// TwinCAT 3 PLC project HomePLC_AlarmManager
// Title: HomePLC Alarm Manager
// Company: Tom Oyen
// Author: Tom Oyen
// ProjectVersion: 1.0.5
// Description: Alarm manager
// ProgramVersion: 3.1.4024.0
// libraries:
//   HomePLC DIO, * (Tom Oyen)
//   HomePLC Logging, * (Tom Oyen)
//   Tc2_Standard, * (Beckhoff Automation GmbH)
//   Tc2_System, * (Beckhoff Automation GmbH)
//   Tc2_Utilities, * (Beckhoff Automation GmbH)
//   Tc3_Module, * (Beckhoff Automation GmbH)
// project tree:
//   DUTs/ E_AlarmManagerStep.TcDUT, E_AlarmState.TcDUT, ST_AlarmManagerHMI.TcDUT
//   / GlobalTextList.TcGTLO, Visualization Manager.TcVMO (not stored)
//   GVLs/ GVL_AlarmManager.TcGVL
//   POUs/ FB_AlarmManager.TcPOU, I_AlarmManager.TcIO
//   POUs/Keypad/DUTs/ E_KeypadState.TcDUT, ST_AlarmKeypadHMI.TcDUT, ST_AlarmKeypadVirtual.TcDUT, ST_LedState.TcDUT
//   POUs/Keypad/ FB_AlarmKeypad.TcPOU, I_AlarmKeypad.TcIO
//   POUs/Sensor/DUTs/ ST_AlarmSensorHMI.TcDUT
//   POUs/Sensor/ FB_AlarmSensor.TcPOU, I_AlarmSensor.TcIO
//   POUs/Siren/DUTs/ ST_AlarmSirenHMI.TcDUT
//   POUs/Siren/ FB_AlarmSiren.TcPOU, I_AlarmSiren.TcIO
//   Project Information/ F_GetCompany.TcPOU, F_GetTitle.TcPOU, F_GetVersion.TcPOU
//   UTIL/ GetDateTime.TcPOU
//   Version/ Global_Version.TcGVL
//   VISUs/ Alarm.TcVIS, Keypad.TcVIS, Siren.TcVIS, Sensor.TcVIS

// ---- DUTs/E_AlarmManagerStep.TcDUT
{attribute 'qualified_only'}
{attribute 'strict'}
TYPE E_AlarmManagerStep :
(
	Init 					:= 0,
	CheckEnable				:= 1,
	
	HardwareCheck			:= 10,
	Enabling				:= 11,
	Enable					:= 12,
	
	CheckSensors			:= 20,
	
	Warn					:= 30,
	WaitForDisableWarn		:= 31,
	SoundAlarm				:= 32,
	WaitForDisableAlarm		:= 33,
	
	Disabling				:= 40,
	Disable					:= 41,
	
	Reset					:= 50
);
END_TYPE

// ---- DUTs/E_AlarmState.TcDUT
{attribute 'qualified_only'}
{attribute 'strict'}
{attribute 'to_string'}
TYPE E_AlarmState :
(
	Off 			:= 0,
	Enabling		:= 1,
	Enabled			:= 2,
	Warning			:= 3,
	Tripped			:= 4,
	Disabling		:= 5
);
END_TYPE

// ---- DUTs/ST_AlarmManagerHMI.TcDUT
TYPE ST_AlarmManagerHMI :
STRUCT
	// General
	nKeypads		: INT;				// Number of keypads
	nSensors		: INT;				// Number of sensors
	nSirens			: INT;				// Number of sirens
	eState			: E_AlarmState;		// Alarm enabled state
	nActiveID		: INT;				// ID of alarm component which was last active
	nActiveReason	: INT;				// Reason why alarm component was active
	
	// Overview
	aSensors		: ARRAY [0..GVL_AlarmManager.nMaxSensors - 1] OF ST_AlarmSensorHMI;
	aSirens			: ARRAY [0..GVL_AlarmManager.nMaxSirens - 1] OF ST_AlarmSirenHMI;
END_STRUCT
END_TYPE

// ---- POUs/Keypad/DUTs/E_KeypadState.TcDUT
{attribute 'qualified_only'}
{attribute 'strict'}
TYPE E_KeypadState :
(
	Init 				:= 0,
	Idle				:= 1,
	InputDetected		:= 2,
	CheckInput			:= 3,
	Reset				:= 4	
);
END_TYPE

// ---- POUs/Keypad/DUTs/ST_AlarmKeypadHMI.TcDUT
TYPE ST_AlarmKeypadHMI :
STRUCT
	sName			: STRING;
	
	bLed1			: BOOL;
	bLed2			: BOOL;
	bLed3			: BOOL;
	bLed4			: BOOL;
	bLed5			: BOOL;
	bLed6			: BOOL;
	
	bBuzzer			: BOOL;
	
	sCode			: STRING;
END_STRUCT
END_TYPE

// ---- POUs/Keypad/DUTs/ST_AlarmKeypadVirtual.TcDUT
TYPE ST_AlarmKeypadVirtual :
STRUCT
	bButton1			: BOOL;
	bButton2			: BOOL;
	bButton3			: BOOL;
	bButton4			: BOOL;
	bButton5			: BOOL;
	bButton6			: BOOL;
END_STRUCT
END_TYPE

// ---- POUs/Keypad/DUTs/ST_LedState.TcDUT
TYPE ST_LedState :
STRUCT
	eLed1	: E_DOCommand;
	eLed2	: E_DOCommand;
	eLed3	: E_DOCommand;
	eLed4	: E_DOCommand;
	eLed5	: E_DOCommand;
	eLed6	: E_DOCommand;
END_STRUCT
END_TYPE

// ---- POUs/Sensor/DUTs/ST_AlarmSensorHMI.TcDUT
TYPE ST_AlarmSensorHMI :
STRUCT
	sName		: STRING;	// Sensor name
	nID			: INT;		// Alarm component ID
	bAlarm		: BOOL;		// True if the sensor detects something
	bTamper		: BOOL;		// True if the sensor is tampered with
	bDisabled	: BOOL;		// True if the sensor is disabled
END_STRUCT
END_TYPE

// ---- POUs/Siren/DUTs/ST_AlarmSirenHMI.TcDUT
TYPE ST_AlarmSirenHMI :
STRUCT
	sName		: STRING;	// Siren name
	nID			: INT;		// Alarm component ID
	bSiren		: BOOL;		// True if the siren is on
	bLight		: BOOL;		// True if the light is on
	bTamper		: BOOL;		// True if the siren is tampered with
END_STRUCT
END_TYPE

// ---- GVLs/GVL_AlarmManager.TcGVL
{attribute 'qualified_only'}
VAR_GLOBAL CONSTANT
	nMaxKeypads		: INT := 5;										// Maximum number of keypads
	nMaxSirens		: INT := 5;										// Maximum number of sirens
	nMaxSensors		: INT := 10;									// Maximum number of sensors
	sCode			: STRING := '1234';								// Configured alarm code
END_VAR

// ---- Version/Global_Version.TcGVL
{attribute 'TcGenerated'}
{attribute 'no-analysis'}
{attribute 'linkalways'}
// This function has been automatically generated from the project information.
VAR_GLOBAL CONSTANT
	{attribute 'const_non_replaced'}
	stLibVersion_HomePLC_Alarm_Manager : ST_LibVersion := (iMajor := 1, iMinor := 0, iBuild := 5, iRevision := 0, nFlags := 0, sVersion := '1.0.5');
END_VAR

// ---- POUs/I_AlarmManager.TcIO
// Alarm manager interface
INTERFACE I_AlarmManager

// Add a keypad to the alarm manager
METHOD AddKeypad
VAR_INPUT
	IKeypad		: I_AlarmKeypad;		// Keypad interface
END_VAR
END_METHOD

// Add an alarm sensor to the alarm manager
METHOD AddSensor
VAR_INPUT
	ISensor		: I_AlarmSensor;		// Alarm sensor interface
END_VAR
END_METHOD

// Add a siren to the alarm manager
METHOD AddSiren
VAR_INPUT
	ISiren		: I_AlarmSiren;		// Siren interface
END_VAR
END_METHOD

END_INTERFACE

// ---- POUs/Keypad/I_AlarmKeypad.TcIO
// Alarm keypad interface
INTERFACE I_AlarmKeypad

// Returns true if the user input code equals the configured code
METHOD CheckCode : BOOL
END_METHOD

// Run this method every cycle
METHOD Execute
END_METHOD

// Returns the HMI data
PROPERTY HmiData : ST_AlarmKeypadHMI
GET
END_GET
END_PROPERTY

// Returns the keypad name
PROPERTY Name : STRING
GET
END_GET
END_PROPERTY

// Call this method once when the alarm state is changed
METHOD SetAlarmState
VAR_INPUT
	eAlarmState			: E_AlarmState;		// Alarm state
END_VAR
END_METHOD

// Set the buzzer command
METHOD SetBuzzer
VAR_INPUT
	eCommand	: E_DOCommand;
END_VAR
END_METHOD

// Set the keypad configured code
METHOD SetConfiguredCode
VAR_INPUT
	sCode	:	STRING;		// Configured code
END_VAR
END_METHOD

// Returns true if the buzzer needs to sound to indicate the alarm status
PROPERTY SoundBuzzer : BOOL
GET
END_GET
END_PROPERTY

END_INTERFACE

// ---- POUs/Sensor/I_AlarmSensor.TcIO
// Alarm sensor interface
INTERFACE I_AlarmSensor

// Returns true if the sensor detects something (as long as something is detected)
PROPERTY Alarm : BOOL
GET
END_GET
END_PROPERTY

// Returns true when the sensor is triggered (one cycle)
PROPERTY AlarmTrigger : BOOL
GET
END_GET
END_PROPERTY

// Run this method every cycle
METHOD Execute
END_METHOD

// Returns the HMI data
PROPERTY HmiData : ST_AlarmSensorHMI
GET
END_GET
END_PROPERTY

// Get the alarm component ID of the sensor
PROPERTY ID : INT
GET
END_GET
END_PROPERTY

// Gets the outputs to turn on when the sensor is triggered
PROPERTY OutputsOnDetect : ARRAY [0..9] OF I_DigitalOut
GET
END_GET
END_PROPERTY

// Number of outputs to enable when the sensor is triggered
PROPERTY OutputsOnDetectSize : INT
GET
END_GET
END_PROPERTY

// Set the sensor disable state
METHOD SetDisableState
VAR_INPUT
	bDisable	: BOOL;		// Set to true to disable the sensor
END_VAR
END_METHOD

// Returns true when the sensor is tampered with (as long as the sensor is tampered with)
PROPERTY Tamper : BOOL
GET
END_GET
END_PROPERTY

// Returns true when the tamper sensor is triggered (one cycle)
PROPERTY TamperTrigger : BOOL
GET
END_GET
END_PROPERTY

// Returs true if the user is warned before the alarm is set off
PROPERTY WarnFirst : BOOL
GET
END_GET
END_PROPERTY

END_INTERFACE

// ---- POUs/Siren/I_AlarmSiren.TcIO
INTERFACE I_AlarmSiren

// Run this method every cycle
METHOD Execute
END_METHOD

// Returns the HMI data
PROPERTY HmiData : ST_AlarmSirenHMI
GET
END_GET
END_PROPERTY

// Get the alarm component ID of the siren
PROPERTY ID : INT
GET
END_GET
END_PROPERTY

// Set siren light
METHOD SetLight
VAR_INPUT
	eCommand	: E_DOCommand;		// Siren digital output command
END_VAR
END_METHOD

// Set siren sound
METHOD SetSound
VAR_INPUT
	eCommand	: E_DOCommand;		// Siren sound digital output command
END_VAR
END_METHOD

// Returns true when the siren is tampered with (as long as the siren is tampered with)
PROPERTY Tamper : BOOL
GET
END_GET
END_PROPERTY

// Returns true when the tamper sensor is triggered (one cycle)
PROPERTY TamperTrigger : BOOL
GET
END_GET
END_PROPERTY

END_INTERFACE

// ---- POUs/FB_AlarmManager.TcPOU
// Alarm manager
{attribute 'reflection'} 
FUNCTION_BLOCK FB_AlarmManager IMPLEMENTS I_AlarmManager
VAR
	aKeypads				: ARRAY [0..GVL_AlarmManager.nMaxKeypads - 1] OF I_AlarmKeypad;		// Keypads
	nKeypads				: INT;																// Number of keypads
	
	aSensors				: ARRAY [0..GVL_AlarmManager.nMaxSensors - 1] OF I_AlarmSensor;		// Alarm sensors
	nSensors				: INT;																// Number of alarm sensors
	
	aSirens					: ARRAY [0..GVL_AlarmManager.nMaxSirens - 1] OF I_AlarmSiren;		// Alarm sirens
	nSirens					: INT;																// Number of alarm sirens
	
	eState					: E_AlarmState;														// Alarm state
	
	bEnabling		AT %Q*	: BOOL;																// Alarm enabling (can be read externally)
	bEnabled		AT %Q*	: BOOL;																// Alarm enabled (can be read externally)
	nState			AT %Q*	: INT;																// Alarm state number (can be read externally)
	nActiveID		AT %Q*	: INT;																// Alarm component ID that tripped alarm (can be read externally)
	nActiveReason	AT %Q*	: INT;																// ID reason alarm was tripped (can be read externally)
	
	fbLogger				: class_Tc3EventLogger;												// Logging FB

	// Use attributes to copy instance name to sName
	{attribute 'instance-path'} 
    {attribute 'noinit'} 
    sName					: STRING; 															// Instance name
	
	stHMI					: ST_AlarmManagerHMI;												// HMI data
END_VAR

// Add a keypad to the alarm manager
METHOD AddKeypad
VAR_INPUT
	IKeypad		: I_AlarmKeypad;		// Keypad interface
END_VAR
// Add keypad
aKeypads[nKeypads] := IKeypad;
nKeypads := nKeypads + 1;
END_METHOD

// Add an alarm sensor to the alarm manager
METHOD AddSensor
VAR_INPUT
	ISensor		: I_AlarmSensor;		// Alarm sensor interface
END_VAR
// Add alarm sensor
aSensors[nSensors] := ISensor;
nSensors := nSensors + 1;
END_METHOD

// Add a siren to the alarm manager
METHOD AddSiren
VAR_INPUT
	ISiren		: I_AlarmSiren;		// Siren interface
END_VAR
// Add siren
aSirens[nSirens] := ISiren;
nSirens := nSirens + 1;
END_METHOD

// Run this method every cycle
METHOD Execute
VAR_INST
	eStep						: E_AlarmManagerStep;	// Alarm manager state machine step
	eStepPrev					: E_AlarmManagerStep;	// Alarm manager state machine previous step
	bFirstCall					: BOOL;					// Alarm manager state machine step first call
	
	bCodeEntered				: BOOL;					// True if the configured code was entered on a keypad
	bSoundBuzzer				: BOOL;					// True if the buzzer needs to sound to indicate the alarm status
	bEnablingBuzzer				: BOOL;					// True if the buzzer needs to sound when enabling the alarm
	bResetSensors				: BOOL;					// True if the sensor disable states need to be reset
	bSensorTriggered			: BOOL;					// True if a sensor is triggered
	bSensorTampered				: BOOL;					// True if a sensor is tampered with
	bWarn						: BOOL;					// True if the user needs to be warned first when a sensor is triggered
	aOutputOnDetect				: ARRAY [0..9] OF I_DigitalOut;	// Returns the outputs to turn on when the sensor is triggered
	nOutputOnDetect				: INT;					// Returns the number of outputs in aOutputOnDetect
	bSirenTampered				: BOOL;					// True if a siren is tampered with
	nActiveSensorID				: INT;					// Alarm component ID of activated sensor
	nActiveSirenID				: INT;					// Alarm component ID of tampered siren
	
	eBuzzerCommand				: E_DOCommand;			// Keypad buzzer digital output command
	eSirenLightCommand			: E_DOCommand;			// Siren light digital output command
	eSirenSoundCommand			: E_DOCommand;			// Siren sound digital output command
	
	fbTimer						: TON;					// Timer FB
	
	sLog						: STRING;				// Log string
END_VAR
VAR
	i							: INT;					// Iterator variable
END_VAR
// Execute methods
Execute_Keypads(eBuzzerCommand := eBuzzerCommand,
				bCodeEntered => bCodeEntered,
				bSoundBuzzer => bSoundBuzzer);
Execute_Sensors(bResetDisableStates := bResetSensors,
				bSensorTriggered => bSensorTriggered,
				bSensorTampered => bSensorTampered,
				bWarn => bWarn,
				nActiveSensorID => nActiveSensorID,
				oaOutputOnDetect => aOutputOnDetect,
				onOutputOnDetect => nOutputOnDetect);
Execute_Sirens(eLightCommand := eSirenLightCommand,
				eSoundCommand := eSirenSoundCommand,
				bSirenTampered => bSirenTampered,
				nActiveSirenID => nActiveSirenID);

// Set variables
bFirstCall := eStep <> eStepPrev;
eStepPrev := eStep;

// Execute alarm logic
CASE eStep OF
	E_AlarmManagerStep.Init:
		// Initialize
		eStep := E_AlarmManagerStep.CheckEnable;
		
	E_AlarmManagerStep.CheckEnable:
		// Check if configured code is entered by the user
		IF bCodeEntered THEN
			// Reset variables
			nActiveID := 0;
			nActiveReason := 0;
			
			// Reset sensor disabled states
			bResetSensors := TRUE;
			
			// Save whether to sound buzzer during enabling
			bEnablingBuzzer := bSoundBuzzer;
			
			eStep := E_AlarmManagerStep.HardwareCheck;
		END_IF
		
	E_AlarmManagerStep.HardwareCheck:
		// Hardware check before enabling alarm
		
		// Check if a sensor detects something or if one is tampered with
		// Check if a siren is tampered with
		IF bSensorTampered OR bSirenTampered THEN
			// Sound buzzer to indicate alarm cannot be enabled
			eBuzzerCommand := E_DOCommand.Flash;
			
			fbLogger.AddInfo('Alarm cannot be enabled due to tampering');
			
			eStep := E_AlarmManagerStep.Reset;
		ELSE
			eStep := E_AlarmManagerStep.Enabling;
		END_IF
		
	E_AlarmManagerStep.Enabling:
		// Enabling alarm
		IF bFirstCall THEN
			// Initialize timer
			fbTimer.PT := T#20S;
			fbTimer(IN := FALSE);
			
			// Set alarm state
			eState := E_AlarmState.Enabling;
			
			// Check if the buzzer needs to be used when enabling the alarm
			IF bEnablingBuzzer THEN
				// Set buzzer to blinking
				eBuzzerCommand := E_DOCommand.Blink;
			END_IF
		ELSE
			// Run timer FB
			fbTimer(IN := TRUE);
			
			// Check if timer expired
			IF fbTimer.Q THEN
				// Turn off buzzer
				eBuzzerCommand := E_DOCommand.Off;
			
				eStep := E_AlarmManagerStep.Enable;
			END_IF
		END_IF
		
		// Check if configure code is entered by user
		IF bCodeEntered THEN
			eStep := E_AlarmManagerStep.Disabling;
		END_IF
	
	E_AlarmManagerStep.Enable:
		// Enable alarm
		eState := E_AlarmState.Enabled;
		
		fbLogger.AddInfo('Alarm enabled');
		
		eStep := E_AlarmManagerStep.CheckSensors;
		
	E_AlarmManagerStep.CheckSensors:
		// Check if configure code is entered by user
		IF bCodeEntered THEN
			eStep := E_AlarmManagerStep.Disabling;
		END_IF
		
		// Check if a sensor or siren is tampered with
		IF bSensorTampered OR bSirenTampered THEN
			// Save what tripped alarm
			nActiveReason := 1;		// Tampering
			
			IF bSensorTampered THEN
				nActiveID := nActiveSensorID;
			END_IF
			
			IF bSirenTampered THEN
				nActiveID := nActiveSirenID;
			END_IF
			
			sLog := CONCAT('Alarm tripped because of tampering by ID ', TO_STRING(nActiveID));
			fbLogger.AddWarning(sLog);
			
			eStep := E_AlarmManagerStep.SoundAlarm;
		END_IF
		
		// Check if a sensor detects something
		IF bSensorTriggered THEN
			// Save sensor name
			nActiveID := nActiveSensorID;
			nActiveReason := 2;		// Motion
			
			sLog := CONCAT('Alarm tripped because of motion by ID ', TO_STRING(nActiveID));
			fbLogger.AddWarning(sLog);
			
			// Check if user needs to be warned
			IF bWarn THEN
				eStep := E_AlarmManagerStep.Warn;
			ELSE				
				eStep := E_AlarmManagerStep.SoundAlarm;
			END_IF
		END_IF
		
	E_AlarmManagerStep.Warn:
		// Warn the user before sounding the alarm
		eBuzzerCommand := E_DOCommand.On;
		
		// Set alarm state
		eState := E_AlarmState.Warning;
		
		fbLogger.AddInfo('Sensor triggered, warning user');
		
		eStep := E_AlarmManagerStep.WaitForDisableWarn;
		
	E_AlarmManagerStep.WaitForDisableWarn:
		// Wait for user to disable alarm and sound the alarm if it does not happen in time
		IF bFirstCall THEN
			// Initialize timer
			fbTimer.PT := T#30S;
			fbTimer(IN := FALSE);
		ELSE
			// Run timer FB
			fbTimer(IN := TRUE);
			
			// Check if configured code is entered by user
			IF bCodeEntered THEN
				// Disable alarm
				eStep := E_AlarmManagerStep.Disabling;
			END_IF
			
			// Check if timer expired
			IF fbTimer.Q THEN
				// Sound alarm
				eStep := E_AlarmManagerStep.SoundAlarm;
			END_IF
		END_IF
		
	E_AlarmManagerStep.SoundAlarm:
		// Turn on alarm sound
		eSirenSoundCommand := E_DOCommand.On;
		
		// Set alarm state
		eState := E_AlarmState.Tripped;
		
		// Turn off buzzer (if on)
		eBuzzerCommand := E_DOCommand.Off;
		
		// Turn on digital outputs associated with sensor that was triggered
		IF nOutputOnDetect > 0 THEN
			FOR i := 0 TO nOutputOnDetect - 1 DO
				aOutputOnDetect[i].SetCommand(eCommandIn := E_DOCommand.On);
			END_FOR
		END_IF
		
		fbLogger.AddInfo('Sounding alarm');
		
		eStep := E_AlarmManagerStep.WaitForDisableAlarm;
		
	E_AlarmManagerStep.WaitForDisableAlarm:
		// Wait for user to disable alarm or wait some time before turning it off automatically
		IF bFirstCall THEN
			// Initialize timer
			fbTimer.PT := T#3M;
			fbTimer(IN := FALSE);
		ELSE
			// Run timer FB
			fbTimer(IN := TRUE);
			
			// Check if configured code is entered by user or if timer expired
			IF bCodeEntered OR fbTimer.Q THEN
				// Disable alarm
				eStep := E_AlarmManagerStep.Disabling;
			END_IF
		END_IF
		
	E_AlarmManagerStep.Disabling:
		IF bFirstCall THEN
			// Turn off alarm sound
			eSirenSoundCommand := E_DOCommand.Off;
		
			// Turn off buzzer (if on)
			eBuzzerCommand := E_DOCommand.Off;
			
			// Set alarm status
			eState := E_AlarmState.Disabling;
			
			// Initialize timer
			fbTimer.PT := T#1.5S;
			fbTimer(IN := FALSE);
		ELSE
			// Run timer FB
			fbTimer(IN := TRUE);
			
			// Check if timer expired
			IF fbTimer.Q THEN
				// Disable alarm
				eStep := E_AlarmManagerStep.Disable;
			END_IF
		END_IF
		
	E_AlarmManagerStep.Disable:
		// Set alarm status
		eState := E_AlarmState.Off;
		
		fbLogger.AddInfo('Alarm disabled');
		
		eStep := E_AlarmManagerStep.Reset;
		
	E_AlarmManagerStep.Reset:
		eStep := E_AlarmManagerStep.CheckEnable;
		
END_CASE

// Update variables
nState := eState;
bEnabling := eState = E_AlarmState.Enabling;
bEnabled := eState = E_AlarmState.Enabled;

// Update HMI
UpdateHMI();
END_METHOD

// Run this method every cycle
METHOD PRIVATE Execute_Keypads
VAR_INPUT
	eBuzzerCommand			: E_DOCommand;	// Keypad buzzer command
END_VAR
VAR_OUTPUT
	bCodeEntered			: BOOL;			// Returns true if the configured code is entered by the user
	bSoundBuzzer			: BOOL;			// Returns true if the buzzer needs to sound to indicate the alarm status
END_VAR
VAR_INST
	bInit					: BOOL;			// Initialized flag
	eBuzzerCommandPrev		: E_DOCommand;	// Previous buzzer digital output command
	fbBuzzerCommandTrigger	: R_TRIG;		// Buzzer command trigger
	eStatePrev				: E_AlarmState;	// Previous alarm state
	fbStateTrigger			: R_TRIG;		// Alarm state change trigger
END_VAR
VAR
	i						: INT;			// Iterator variable
END_VAR
// Check if buzzer command changed
fbBuzzerCommandTrigger(CLK := eBuzzerCommand <> eBuzzerCommandPrev);
eBuzzerCommandPrev := eBuzzerCommand;

// Check if alarm state changed
fbStateTrigger(CLK := eState <> eStatePrev);
eStatePrev := eState;

// Initialize variable
bCodeEntered := FALSE;

FOR i := 0 TO nKeypads - 1 DO	
	// Set keypad configure code
	aKeypads[i].SetConfiguredCode(sCode := GVL_AlarmManager.sCode);
	
	// Check if buzzer command changed
	IF fbBuzzerCommandTrigger.Q THEN
		// Set buzzer digital output command
		aKeypads[i].SetBuzzer(eCommand := eBuzzerCommand);
	END_IF
	
	// Check if alarm state changed
	IF fbStateTrigger.Q OR NOT bInit THEN
		// Update keypad on alarm state change
		aKeypads[i].SetAlarmState(eAlarmState := eState);
	END_IF
	
	// Run keypad Execute method
	aKeypads[i].Execute();
	
	// Check if the configured code is entered on at least one keypad
	IF aKeypads[i].CheckCode() THEN
		bCodeEntered := TRUE;
		bSoundBuzzer := aKeypads[i].SoundBuzzer;
	END_IF
END_FOR

bInit := TRUE;
END_METHOD

// Run this method every cycle
METHOD PRIVATE Execute_Sensors
VAR_INPUT
	bResetDisableStates	: BOOL;					// Set to true to reset all sensor disabled states
END_VAR
VAR_OUTPUT
	bSensorTriggered	: BOOL;					// Returns true if a sensor detects something
	bSensorTampered		: BOOL;					// Returns true if a sensor is tampered with
	bWarn				: BOOL;					// Returns true if a warning is issued first instead of immediately sounding the alarm (only valid on sensor trigger)
	nActiveSensorID		: INT;					// Returns the ID of the active sensor
	oaOutputOnDetect	: ARRAY [0..9] OF I_DigitalOut;	// Returns the outputs to turn on when the sensor is triggered
	onOutputOnDetect	: INT;					// Returns the number of outputs in aOutputOnDetect
END_VAR
VAR_INST
	fbResetTrigger		: R_TRIG;				// Reset disabled state trigger
	aOutputOnDetect		: ARRAY [0..9] OF I_DigitalOut;	// Returns the outputs to turn on when the sensor is triggered
	nOutputOnDetect		: INT;					// Returns the number of outputs in aOutputOnDetect
END_VAR
VAR
	i					: INT;					// Iterator variable
END_VAR
// Initialize variables
bSensorTriggered := FALSE;
bSensorTampered	:= FALSE;
bWarn := TRUE;

// Check reset command
fbResetTrigger(CLK := bResetDisableStates);

FOR i := 0 TO nSensors -1 DO
	// Reset disables states
	IF fbResetTrigger.Q THEN
		aSensors[i].SetDisableState(bDisable := FALSE);
	END_IF

	// Run sensor Execute method
	aSensors[i].Execute();

	// Check if at least one sensor detects something or is tampered with
	bSensorTriggered := bSensorTriggered OR aSensors[i].AlarmTrigger;
	bSensorTampered := bSensorTampered OR aSensors[i].TamperTrigger;
	
	// Check if alarm needs to be sounded immediately or if a warning can be issued first
	IF aSensors[i].AlarmTrigger AND NOT aSensors[i].TamperTrigger THEN
		// Sensor detects something but is not tampered with
		// Warn if the sensor allows a warning
		// If one sensor does not allow a warning, sound the alarm immediately
		bWarn := bWarn AND aSensors[i].WarnFirst;
	END_IF
	
	// Report which sensor was activated
	IF aSensors[i].AlarmTrigger OR aSensors[i].TamperTrigger THEN
		IF nActiveSensorID = 0 THEN
			nActiveSensorID := aSensors[i].ID;
			aOutputOnDetect := aSensors[i].OutputsOnDetect;
			nOutputOnDetect := aSensors[i].OutputsOnDetectSize;
		END_IF
	END_IF
END_FOR

// Set outputs
oaOutputOnDetect := aOutputOnDetect;
onOutputOnDetect := nOutputOnDetect;
END_METHOD

// Run this method every cycle
METHOD PRIVATE Execute_Sirens
VAR_INPUT
	eLightCommand				: E_DOCommand;		// Siren light digital output command
	eSoundCommand				: E_DOCommand;		// Siren sound digital output command
END_VAR
VAR_OUTPUT
	bSirenTampered				: BOOL;				// Returns true if the siren is tampered with
	nActiveSirenID				: INT;				// Returns the name of the tampered siren
END_VAR
VAR
	i							: INT;				// Iterator variable
END_VAR
VAR_INST
	eLightCommandPrev			: E_DOCommand;		// Siren light previous digital output command
	fbLightCommandTrigger		: R_TRIG;			// Siren light command changed trigger
	
	eSoundCommandPrev			: E_DOCommand;		// Siren sound previous digital output command
	fbSoundCommandTrigger		: R_TRIG;			// Siren sound command changed trigger
END_VAR
// Check if the siren light digital command has changed
fbLightCommandTrigger(CLK := eLightCommand <> eLightCommandPrev);
eLightCommandPrev := eLightCommand;

// Check if the siren sound digital command has changed
fbSoundCommandTrigger(CLK := eSoundCommand <> eSoundCommandPrev);
eSoundCommandPrev := eSoundCommand;

// Initialize variable
bSirenTampered	:= FALSE;

FOR i := 0 TO nSirens - 1 DO
	// Check if siren light command changed
	IF fbLightCommandTrigger.Q THEN
		// Set siren light digital output command
		aSirens[i].SetLight(eCommand := eLightCommand);
	END_IF
	
	// Check if siren sound command changed
	IF fbSoundCommandTrigger.Q THEN
		// Set siren sound digital output command
		aSirens[i].SetSound(eCommand := eSoundCommand);
	END_IF
	
	// Run siren Execute method
	aSirens[i].Execute();
	
	// Check if at least one siren is tampered with
	bSirenTampered := bSirenTampered OR aSirens[i].TamperTrigger;
	
	// Report which siren was tampered with
	IF aSirens[i].TamperTrigger THEN
		IF nActiveSirenID = 0 THEN
			nActiveSirenID := aSirens[i].ID;
		END_IF
	END_IF
END_FOR
END_METHOD

// Initialize the alarm manager FB
METHOD FB_init : BOOL
VAR_INPUT
	bInitRetains : BOOL; // if TRUE, the retain variables are initialized (warm start / cold start)
	bInCopyCode : BOOL;  // if TRUE, the instance afterwards gets moved into the copy code (online change)
END_VAR
// Initialize logger
fbLogger.Init(sSource := sName, bEnableVerbose := TRUE);
END_METHOD

// Update HMI
METHOD PRIVATE UpdateHMI
VAR
	i	: INT;	// Iterator variable
END_VAR
// General
stHMI.nKeypads := nKeypads;
stHMI.nSensors := nSensors;
stHMI.nSirens := nSirens;
stHMI.eState := eState;
stHMI.nActiveID := nActiveID;
stHMI.nActiveReason := nActiveReason;

// Overview
FOR i := 0 TO nSensors - 1 DO
	stHMI.aSensors[i] := aSensors[i].HmiData;
END_FOR

FOR i := 0 TO nSirens - 1 DO
	stHMI.aSirens[i] := aSirens[i].HmiData;
END_FOR
END_METHOD

END_FUNCTION_BLOCK

// ---- POUs/Keypad/FB_AlarmKeypad.TcPOU
// Alarm keypad FB (B11-11-11L11-11-11)
FUNCTION_BLOCK FB_AlarmKeypad IMPLEMENTS I_AlarmKeypad
VAR
	sName			: STRING;				// Keypad name
	bSoundBuzzer	: BOOL;					// True if the buzzer should be used to indicate the alarm status when using this keypad

	fbButton1		: FB_DigitalIn;			// Button 1
	fbLed1			: FB_DigitalOut;		// LED 1
	fbButton2		: FB_DigitalIn;			// Button 2
	fbLed2			: FB_DigitalOut;		// LED 2
	fbButton3		: FB_DigitalIn;			// Button 3
	fbLed3			: FB_DigitalOut;		// LED 3
	fbButton4		: FB_DigitalIn;			// Button 4
	fbLed4			: FB_DigitalOut;		// LED 4
	fbButton5		: FB_DigitalIn;			// Button 5
	fbLed5			: FB_DigitalOut;		// LED 5
	fbButton6		: FB_DigitalIn;			// Button 6
	fbLed6			: FB_DigitalOut;		// LED 6
	fbBuzzer		: FB_DigitalOut;		// Buzzer

	eState			: E_KeypadState;		// Keypad state
	sConfiguredCode	: STRING;				// Configured alarm code
	sInputCode		: STRING;				// User input code
	dtInputTime		: DATE_AND_TIME;		// Date and time of last user input
	stLedsDefault	: ST_LedState;			// Default LEDs state
	
	stHMI			: ST_AlarmKeypadHMI;	// HMI data
	stVirtual		: ST_AlarmKeypadVirtual;	// Virtual keypad
END_VAR

// Returns true if the user input code equals the configured code
METHOD CheckCode : BOOL
// Compare codes
CheckCode := sInputCode = sConfiguredCode;

// Reset input if correct code was entered
IF CheckCode THEN
	Reset();
END_IF
END_METHOD

// Collect user input from buttons and build the entered code, returns true if input was detected
METHOD PRIVATE CollectInput: BOOL
VAR
	sInput			: STRING;
END_VAR
// Check buttons and translate to input
IF fbButton1.Command = E_DICommand.ShortPress THEN sInput := '1'; END_IF
IF fbButton2.Command = E_DICommand.ShortPress THEN sInput := '2'; END_IF
IF fbButton3.Command = E_DICommand.ShortPress THEN sInput := '3'; END_IF
IF fbButton4.Command = E_DICommand.ShortPress THEN sInput := '4'; END_IF
IF fbButton5.Command = E_DICommand.ShortPress THEN sInput := '5'; END_IF
IF fbButton6.Command = E_DICommand.ShortPress THEN sInput := '6'; END_IF

// Check if input was detected
IF sInput <> '' THEN
	// Build user input code
	sInputCode := CONCAT(sInputCode, sInput);
	
	// Update time of last input
	dtInputTime := GetDateTime();
	
	// Set output
	CollectInput := TRUE;
ELSE
	// Set output
	CollectInput := FALSE;
END_IF
END_METHOD

// Run this method every cycle
METHOD Execute
VAR CONSTANT
	stLedsOn	: ST_LedState := (eLed1 := E_DOCommand.On,
									eLed2 := E_DOCommand.On,
									eLed3 := E_DOCommand.On,
									eLed4 := E_DOCommand.On,
									eLed5 := E_DOCommand.On,
									eLed6 := E_DOCommand.On);
END_VAR
// Keypad state machine
CASE eState OF
	E_KeypadState.Init:
		// Initialize
		eState := E_KeypadState.Idle;
	
	E_KeypadState.Idle:
		// Wait for input
		IF CollectInput() THEN
			eState := E_KeypadState.InputDetected;
		END_IF
	
	E_KeypadState.InputDetected:
		// Collect input in every state so no input is lost
		CollectInput();
		
		// Enable all LEDs
		SetLeds(stLedsOn);
		
		eState := E_KeypadState.CheckInput;
		
	E_KeypadState.CheckInput:
		// Continue collecting input
		CollectInput();
		
		// If no input is detected during some time, reset the keypad
		IF GetDateTime() - dtInputTime > T#2S THEN
			eState := E_KeypadState.Reset;
		END_IF
		
	E_KeypadState.Reset:
		// Reset keypad
		Reset();
		
		eState := E_KeypadState.Idle;
END_CASE

// Update HMI
UpdateHMI();
END_METHOD

METHOD FB_init : BOOL
VAR_INPUT
	bInitRetains	: BOOL;		// if TRUE, the retain variables are initialized (warm start / cold start)
	bInCopyCode		: BOOL;		// if TRUE, the instance afterwards gets moved into the copy code (online change)
	
	sKeypadName		: STRING;	// Keypad name
	bSoundBuzzer	: BOOL;		// Set to true to use the buzzer to indicate the alarm status when using this keypad
END_VAR
sName := sKeypadName;
THIS^.bSoundBuzzer := bSoundBuzzer;

fbBuzzer.SetBlinkPeriod(tPeriod := T#1500MS);
END_METHOD

// Returns the HMI data
PROPERTY HmiData : ST_AlarmKeypadHMI
GET
HmiData := stHMI;
END_GET
END_PROPERTY

// Returns the keypad name
PROPERTY Name : STRING
GET
Name := sName;
END_GET
END_PROPERTY

// Reset the keypad
METHOD PRIVATE Reset
// Reset user input code
sInputCode := '';

// Reset all LEDs to their default value
SetLeds(stLedsDefault);
END_METHOD

// Call this method once when the alarm state is changed
METHOD SetAlarmState
VAR_INPUT
	eAlarmState				: E_AlarmState;		// Alarm state
END_VAR
VAR CONSTANT
	stLedsAlarmOn			: ST_LedState := (eLed1 := E_DOCommand.On,
											eLed2 := E_DOCommand.Off,
											eLed3 := E_DOCommand.Off,
											eLed4 := E_DOCommand.Off,
											eLed5 := E_DOCommand.Off,
											eLed6 := E_DOCommand.Off);
	stLedsAlarmOff			: ST_LedState := (eLed1 := E_DOCommand.Off,
											eLed2 := E_DOCommand.Off,
											eLed3 := E_DOCommand.Off,
											eLed4 := E_DOCommand.Off,
											eLed5 := E_DOCommand.Off,
											eLed6 := E_DOCommand.Off);
	stLedsAlarmEnabling		: ST_LedState := (eLed1 := E_DOCommand.Blink,
											eLed2 := E_DOCommand.Off,
											eLed3 := E_DOCommand.Off,
											eLed4 := E_DOCommand.Off,
											eLed5 := E_DOCommand.Off,
											eLed6 := E_DOCommand.Off);
	stLedsAlarmWarning		: ST_LedState := (eLed1 := E_DOCommand.Blink,
											eLed2 := E_DOCommand.Off,
											eLed3 := E_DOCommand.Off,
											eLed4 := E_DOCommand.Off,
											eLed5 := E_DOCommand.Off,
											eLed6 := E_DOCommand.Off);
	stLedsAlarmTripped		: ST_LedState := (eLed1 := E_DOCommand.Blink,
											eLed2 := E_DOCommand.Off,
											eLed3 := E_DOCommand.Off,
											eLed4 := E_DOCommand.Off,
											eLed5 := E_DOCommand.Off,
											eLed6 := E_DOCommand.Off);
	stLedsAlarmDisabling	: ST_LedState := (eLed1 := E_DOCommand.Blink,
											eLed2 := E_DOCommand.Off,
											eLed3 := E_DOCommand.Off,
											eLed4 := E_DOCommand.Off,
											eLed5 := E_DOCommand.Off,
											eLed6 := E_DOCommand.Off);
END_VAR
// Set LEDs default state
CASE eAlarmState OF
	E_AlarmState.Off:
		// Alarm is off
		stLedsDefault := stLedsAlarmOff;
		
	E_AlarmState.Enabling:
		// Alarm is enabling
		fbLed1.SetBlinkPeriod(tPeriod := T#1500MS);	// Same as buzzer
		stLedsDefault := stLedsAlarmEnabling;
	
	E_AlarmState.Enabled:
		// Alarm is on
		stLedsDefault := stLedsAlarmOn;
		
	E_AlarmState.Warning:
		// Alarm is warning
		fbLed1.SetBlinkPeriod(tPeriod := T#500MS);	// Fast blinking, buzzer is on continuously
		stLedsDefault := stLedsAlarmWarning;
		
	E_AlarmState.Tripped:
		// Alarm has been tripped
		fbLed1.SetBlinkPeriod(tPeriod := T#500MS);	// Fast blinking, alarm is sounding
		stLedsDefault := stLedsAlarmTripped;
		
	E_AlarmState.Disabling:
		// Alarm has been tripped
		fbLed1.SetBlinkPeriod(tPeriod := T#250MS);	// Fast blinking, indicate alarm is disabling
		stLedsDefault := stLedsAlarmDisabling;
END_CASE

// Reset keypad
Reset();
END_METHOD

// Set the buzzer command
METHOD SetBuzzer
VAR_INPUT
	eCommand	: E_DOCommand;
END_VAR
// Set digital output command
fbBuzzer.SetCommand(eCommandIn := eCommand);
END_METHOD

// Set the keypad configured code
METHOD SetConfiguredCode
VAR_INPUT
	sCode	:	STRING;		// Configured code
END_VAR
// Set configured alarm code
sConfiguredCode := sCode;
END_METHOD

// Set the LEDs state
METHOD PRIVATE SetLeds
VAR_INPUT
	stLeds		: ST_LedState;		// LED states
END_VAR
fbLed1.SetCommand(eCommandIn := stLeds.eLed1);
fbLed2.SetCommand(eCommandIn := stLeds.eLed2);
fbLed3.SetCommand(eCommandIn := stLeds.eLed3);
fbLed4.SetCommand(eCommandIn := stLeds.eLed4);
fbLed5.SetCommand(eCommandIn := stLeds.eLed5);
fbLed6.SetCommand(eCommandIn := stLeds.eLed6);
END_METHOD

// Returns true if the buzzer needs to sound to indicate the alarm status
PROPERTY SoundBuzzer : BOOL
GET
SoundBuzzer := bSoundBuzzer;
END_GET
END_PROPERTY

// Update HMI
METHOD PRIVATE UpdateHMI
VAR
	stLed1HMI	: ST_HmiDigitalOut;
	stLed2HMI	: ST_HmiDigitalOut;
	stLed3HMI	: ST_HmiDigitalOut;
	stLed4HMI	: ST_HmiDigitalOut;
	stLed5HMI	: ST_HmiDigitalOut;
	stLed6HMI	: ST_HmiDigitalOut;
	stBuzzerHMI	: ST_HmiDigitalOut;
END_VAR
// Get data
stLed1HMI := fbLed1.HmiData;
stLed2HMI := fbLed2.HmiData;
stLed3HMI := fbLed3.HmiData;
stLed4HMI := fbLed4.HmiData;
stLed5HMI := fbLed5.HmiData;
stLed6HMI := fbLed6.HmiData;
stBuzzerHMI := fbBuzzer.HmiData;

// Set HMI data
stHMI.bLed1 := stLed1HMI.bValue;
stHMI.bLed2 := stLed2HMI.bValue;
stHMI.bLed3 := stLed3HMI.bValue;
stHMI.bLed4 := stLed4HMI.bValue;
stHMI.bLed5 := stLed5HMI.bValue;
stHMI.bLed6 := stLed6HMI.bValue;
stHMI.bBuzzer := stBuzzerHMI.bValue;

stHMI.sCode := sInputCode;
stHMI.sName := sName;

// Set buttons
fbButton1.SetExternalIn(bIn := stVirtual.bButton1);
fbButton2.SetExternalIn(bIn := stVirtual.bButton2);
fbButton3.SetExternalIn(bIn := stVirtual.bButton3);
fbButton4.SetExternalIn(bIn := stVirtual.bButton4);
fbButton5.SetExternalIn(bIn := stVirtual.bButton5);
fbButton6.SetExternalIn(bIn := stVirtual.bButton6);
END_METHOD

END_FUNCTION_BLOCK

// ---- UTIL/GetDateTime.TcPOU
// Gets the current date and time (now)
FUNCTION GetDateTime : DATE_AND_TIME
VAR
	fbSystemTime : GETSYSTEMTIME;
	timeAsFileTime : T_FILETIME;
END_VAR

fbSystemTime(timeLoDW => timeAsFileTime.dwLowDateTime, timeHiDW => timeAsFileTime.dwHighDateTime);
GetDateTime := FILETIME_TO_DT(timeAsFileTime);

END_FUNCTION

// ---- POUs/Sensor/FB_AlarmSensor.TcPOU
// Alarm sensor FB
FUNCTION_BLOCK FB_AlarmSensor IMPLEMENTS I_AlarmSensor
VAR
	sName					: STRING;				// Sensor name
	nID						: INT;					// Alarm component ID
	bWarnFirst				: BOOL;					// Set to true to warn the user before setting off the alarm
	bDisable		AT %I*	: BOOL;					// Set to true to disable the sensor (can be set externally)
	
	ibAlarm			AT %I*	: BOOL;					// Active low alarm input
	ibTamper		AT %I*	: BOOL;					// Active low tamper input
	
	bAlarm					: BOOL;					// True if the sensor detects something
	bTamper					: BOOL;					// True if the sensor is tampered with
	
	bAlarmTrigger			: BOOL;					// Returns true when the sensor is triggered
	bTamperTrigger			: BOOL;					// Returns true when the sensor is tampered with
	
	aOutputOnDetect			: ARRAY [0..9] OF I_DigitalOut;	// Digital outputs to turn on when sensor is triggered
	nOutputOnDetect			: INT;					// Number of digitial outputs in aOutputOnDetect
	
	stHMI					: ST_AlarmSensorHMI;	// HMI data
END_VAR

// Add a digital output to turn on when the sensor is triggered
METHOD AddOutputOnDetect
VAR_INPUT
	IDO		: I_DigitalOut;
END_VAR
aOutputOnDetect[nOutputOnDetect] := IDO;
nOutputOnDetect := nOutputOnDetect + 1;
END_METHOD

// Returns true if the sensor detects something (as long as something is detected)
PROPERTY Alarm : BOOL
GET
Alarm := bAlarm;
END_GET
END_PROPERTY

// Returns true when the sensor is triggered (one cycle)
PROPERTY AlarmTrigger : BOOL
GET
AlarmTrigger := bAlarmTrigger;
END_GET
END_PROPERTY

// Run this method every cycle
METHOD Execute
VAR_INST
	fbAlarm		: R_TRIG;		// Alarm rising trigger
	fbTamper	: R_TRIG;		// Tamper rising trigger
END_VAR
// Check if disabled
IF NOT bDisable THEN
	// Convert active low inputs
	bAlarm := NOT ibAlarm;
	bTamper := NOT ibTamper;
END_IF

// Run FBs
fbAlarm(CLK := bAlarm);
fbTamper(CLK := bTamper);

// Check triggers
bAlarmTrigger := fbAlarm.Q;
bTamperTrigger := fbTamper.Q;

// Update HMI
UpdateHMI();
END_METHOD

METHOD FB_init : BOOL
VAR_INPUT
	bInitRetains	: BOOL;		// if TRUE, the retain variables are initialized (warm start / cold start)
	bInCopyCode		: BOOL;		// if TRUE, the instance afterwards gets moved into the copy code (online change)
	
	sSensorName		: STRING;	// Sensor name
	nSensorID		: INT;		// Sensor ID
	bEnableWarning	: BOOL;		// Set to true to warn the user before setting off the alarm
END_VAR
sName := sSensorName;
nID := nSensorID;
bWarnFirst := bEnableWarning;
END_METHOD

// Returns the HMI data
PROPERTY HmiData : ST_AlarmSensorHMI
GET
HmiData := stHMI;
END_GET
END_PROPERTY

// Get the alarm component ID of the sensor
PROPERTY ID : INT
GET
ID := nID;
END_GET
END_PROPERTY

// Gets the outputs to turn on when the sensor is triggered
PROPERTY OutputsOnDetect : ARRAY [0..9] OF I_DigitalOut
GET
OutputsOnDetect := aOutputOnDetect;
END_GET
END_PROPERTY

// Number of outputs to enable when the sensor is triggered
PROPERTY OutputsOnDetectSize : INT
GET
OutputsOnDetectSize := nOutputOnDetect;
END_GET
END_PROPERTY

// Set the sensor disable state
METHOD SetDisableState
VAR_INPUT
	bDisable	: BOOL;		// Set to true to disable the sensor
END_VAR
THIS^.bDisable := bDisable;
END_METHOD

// Returns true when the sensor is tampered with (as long as the sensor is tampered with)
PROPERTY Tamper : BOOL
GET
Tamper := bTamper;
END_GET
END_PROPERTY

// Returns true when the tamper sensor is triggered (one cycle)
PROPERTY TamperTrigger : BOOL
GET
TamperTrigger := bTamperTrigger;
END_GET
END_PROPERTY

// Update HMI
METHOD PRIVATE UpdateHMI
stHMI.sName := sName;
stHMI.nID := nID;
stHMI.bAlarm := bAlarm;
stHMI.bTamper := bTamper;
stHMI.bDisabled := bDisable;
END_METHOD

// Returs true if the user is warned before the alarm is set off
PROPERTY WarnFirst : BOOL
GET
WarnFirst := bWarnFirst;
END_GET
END_PROPERTY

END_FUNCTION_BLOCK

// ---- POUs/Siren/FB_AlarmSiren.TcPOU
// Alarm siren FB
FUNCTION_BLOCK FB_AlarmSiren IMPLEMENTS I_AlarmSiren
VAR
	sName				: STRING;				// Siren name
	nID					: INT;					// Alarm component ID
	
	ibTamper			AT %I* : BOOL;			// Active low tamper input
	fbLight				: FB_DigitalOut;		// Siren light digital output FB
	fbSiren				: FB_DigitalOut;		// Siren sound digital output FB
	
	bTamper				: BOOL;					// True if the siren is tampered with
	
	bTamperTrigger		: BOOL;					// True when the tamper sensor is triggered (one cycle)
	
	stHMI				: ST_AlarmSirenHMI;		// HMI data
END_VAR

// Run this method every cycle
METHOD Execute
VAR_INST
	fbTamper	: R_TRIG;		// Tamper rising edge
END_VAR
// Convert active low inputs
bTamper := NOT ibTamper;

// Run FBs
fbTamper(CLK := bTamper);

// Check trigger
bTamperTrigger := fbTamper.Q;

// Update HMI
UpdateHMI();
END_METHOD

METHOD FB_init : BOOL
VAR_INPUT
	bInitRetains	: BOOL;		// if TRUE, the retain variables are initialized (warm start / cold start)
	bInCopyCode		: BOOL;		// if TRUE, the instance afterwards gets moved into the copy code (online change)
	
	sSirenName		: STRING;	// Siren name
	nSirenID		: INT;		// Sensor ID
END_VAR
sName := sSirenName;
nID := nSirenID;
END_METHOD

// Returns the HMI data
PROPERTY HmiData : ST_AlarmSirenHMI
GET
HmiData := stHMI;
END_GET
END_PROPERTY

// Get the alarm component ID of the siren
PROPERTY ID : INT
GET
ID := nID;
END_GET
END_PROPERTY

// Set siren light
METHOD SetLight
VAR_INPUT
	eCommand	: E_DOCommand;		// Siren digital output command
END_VAR
// Set siren digital output command
fbLight.SetCommand(eCommandIn := eCommand);
END_METHOD

// Set siren sound
METHOD SetSound
VAR_INPUT
	eCommand	: E_DOCommand;		// Siren sound digital output command
END_VAR
// Set the siren digital output command
fbSiren.SetCommand(eCommandIn := eCommand);
END_METHOD

// Returns true when the siren is tampered with (as long as the siren is tampered with)
PROPERTY Tamper : BOOL
GET
Tamper := bTamper;
END_GET
END_PROPERTY

// Returns true when the tamper sensor is triggered (one cycle)
PROPERTY TamperTrigger : BOOL
GET
TamperTrigger := bTamperTrigger;
END_GET
END_PROPERTY

// Update HMI
METHOD PRIVATE UpdateHMI
VAR
	stSirenHMI	: ST_HmiDigitalOut;
	stLightHMI	: ST_HmiDigitalOut;
END_VAR
// Get data
stSirenHMI := fbSiren.HmiData;
stLightHMI := fbLight.HmiData;

// Set HMI data
stHMI.sName := sName;
stHMI.nID := nID;
stHMI.bSiren := stSirenHMI.bValue;
stHMI.bLight := stLightHMI.bValue;
stHMI.bTamper := bTamper;
END_METHOD

END_FUNCTION_BLOCK

// ---- Project Information/F_GetCompany.TcPOU
// This function has been automatically generated from the project information.
{attribute 'signature_flag' := '1073741824'}
{attribute 'TcGenerated'}
{attribute 'no-analysis'}
FUNCTION F_GetCompany : WSTRING
VAR_INPUT
	
END_VAR

F_GetCompany := "Tom Oyen";

END_FUNCTION

// ---- Project Information/F_GetTitle.TcPOU
// This function has been automatically generated from the project information.
{attribute 'signature_flag' := '1073741824'}
{attribute 'TcGenerated'}
{attribute 'no-analysis'}
FUNCTION F_GetTitle : WSTRING
VAR_INPUT
	
END_VAR

F_GetTitle := "HomePLC Alarm Manager";

END_FUNCTION

// ---- Project Information/F_GetVersion.TcPOU
// This function has been automatically generated from the project information.
{attribute 'signature_flag' := '1073741824'}
{attribute 'TcGenerated'}
{attribute 'no-analysis'}
FUNCTION F_GetVersion : ST_LibVersion
VAR_INPUT
	
END_VAR

F_GetVersion.iMajor := 1;
F_GetVersion.iMinor := 0;
F_GetVersion.iBuild := 5;
F_GetVersion.iRevision := 0;
F_GetVersion.sVersion := '1.0.5';
F_GetVersion.nFlags := 0;

END_FUNCTION

// ---- GlobalTextList.TcGTLO
TEXTLIST GlobalTextList
  756 = '%d'
  426 = '%s'
  221 = '1'
  170 = '2'
  836 = '3'
  541 = '4'
  607 = '5'
  496 = '6'
  182 = 'Alarm'
  950 = 'Buzzer'
  191 = 'Disabled'
  377 = 'ID'
  999 = 'Keypad %s'
  292 = 'Keypads'
  547 = 'Light'
  181 = 'Name'
  693 = 'Sensor %s'
  755 = 'Sensors'
  213 = 'Siren'
  137 = 'Siren %s'
  135 = 'Sirens'
  183 = 'Tamper'
END_TEXTLIST

// ---- VISUs/Alarm.TcVIS
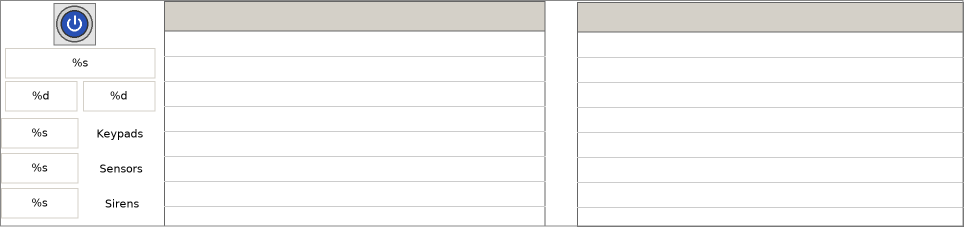
VISUALIZATION Alarm  // 964x227
VAR_IN_OUT
	stAlarm		: ST_AlarmManagerHMI;
END_VAR
    PowerSwitch (50,3 49x42), variable: stAlarm.eState = E_AlarmState.Enabled, input disabled if: TRUE, behaviour: TOGGLE, style: Switch-PowerSwitch-Blue
    Table (164,1 381x225), data array: stAlarm.aSensors
        p3854506369: stAlarm.aSensors[INDEX].sName
        p1892666644: stAlarm.aSensors[INDEX].nID
        p338671338: stAlarm.aSensors[INDEX].bAlarm
        p2170511999: stAlarm.aSensors[INDEX].bTamper
    Table (577,2 387x225), data array: stAlarm.aSirens
        p3854506369: stAlarm.aSirens[INDEX].sName
        p1892666644: stAlarm.aSirens[INDEX].nID
        p338671338: stAlarm.aSirens[INDEX].bSiren
        p2170511999: stAlarm.aSirens[INDEX].bLight
        p3723444502: stAlarm.aSirens[INDEX].bTamper
    Textfield (1,118 77x30), "%s", text variable: stAlarm.nKeypads
    Textfield (1,153 77x30), "%s", text variable: stAlarm.nSensors
    Textfield (1,188 77x30), "%s", text variable: stAlarm.nSirens
    Label (85,119 70x30), "Keypads"
    Label (86,154 70x30), "Sensors"
    Label (87,189 70x30), "Sirens"
    Textfield (5,48 150x30), "%s", text variable: stAlarm.eState
    Textfield (5,81 72x30), "%d", text variable: stAlarm.nActiveID
    Textfield (83,81 72x30), "%d", text variable: stAlarm.nActiveReason
END_VISUALIZATION

// ---- VISUs/Keypad.TcVIS
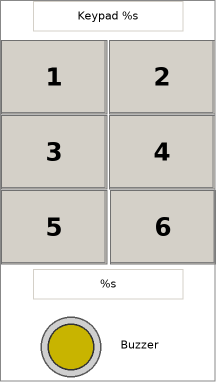
VISUALIZATION Keypad  // 216x382
VAR_IN_OUT
	stKeypadVirtual	: ST_AlarmKeypadVirtual;
	stKeypad		: ST_AlarmKeypadHMI;
END_VAR
    Button (1,40 106x74), "1", colour toggle: stKeypad.bLed1
        tap stKeypadVirtual.bButton1
    Button (109,40 106x74), "2", colour toggle: stKeypad.bLed2
        tap stKeypadVirtual.bButton2
    Button (1,115 106x74), "3", colour toggle: stKeypad.bLed3
        tap stKeypadVirtual.bButton3
    Button (109,115 106x74), "4", colour toggle: stKeypad.bLed4
        tap stKeypadVirtual.bButton4
    Button (1,190 106x74), "5", colour toggle: stKeypad.bLed5
        tap stKeypadVirtual.bButton5
    Button (110,190 106x74), "6", colour toggle: stKeypad.bLed6
        tap stKeypadVirtual.bButton6
    Lamp1 (36,312 70x70), variable: stKeypad.bBuzzer, style: Lamp-Lamp1-Yellow
    Label (115,330 49x30), "Buzzer"
    Textfield (33,269 150x30), "%s", text variable: stKeypad.sCode
    Textfield (33,1 150x30), "Keypad %s", text variable: stKeypad.sName
END_VISUALIZATION

// ---- VISUs/Siren.TcVIS
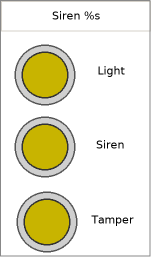
VISUALIZATION Siren  // 151x257
VAR_IN_OUT
	stSiren		: ST_AlarmSirenHMI;
END_VAR
    Lamp1 (10,40 70x70), variable: stSiren.bLight, style: Lamp-Lamp1-Yellow
    Lamp1 (10,112 70x70), variable: stSiren.bSiren, style: Lamp-Lamp1-Yellow
    Label (87,56 49x30), "Light"
    Label (86,130 49x30), "Siren"
    Textfield (1,1 150x30), "Siren %s", text variable: stSiren.sName
    Lamp1 (12,187 70x70), variable: stSiren.bTamper, style: Lamp-Lamp1-Yellow
    Label (88,205 49x30), "Tamper"
END_VISUALIZATION

// ---- VISUs/Sensor.TcVIS
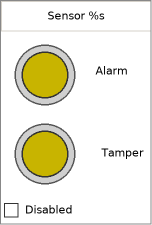
VISUALIZATION Sensor  // 152x225
VAR_IN_OUT
	stSensor		: ST_AlarmSensorHMI;
END_VAR
    Lamp1 (10,40 70x70), variable: stSensor.bAlarm, style: Lamp-Lamp1-Yellow
    Label (87,56 49x30), "Alarm"
    Textfield (1,1 150x30), "Sensor %s", text variable: stSensor.sName
    Lamp1 (10,119 70x70), variable: stSensor.bTamper, style: Lamp-Lamp1-Yellow
    Label (98,138 49x30), "Tamper"
    Checkbox (2,195 150x30), "Disabled", variable: stSensor.bDisabled
END_VISUALIZATION
